Fanuc KAREL source: CURJPOS.kl

PROGRAM T
%NOLOCKGROUP
VAR
 v0 : INTEGER
 v1 : INTEGER
 v2 : INTEGER
 res : JOINTPOS
BEGIN
 res = CURJPOS(v0, v1, v2)
END T
